FUNCTION_BLOCK Test_WhenBusy_Abort_SelectsAborting EXTENDS TUnitTestbase
VAR
END_VAR

METHOD  Execute
VAR
    Execution : TExecution;
END_VAR
Test_Started();

Execution.Start();
Execution.SetBusy();
Execution.Abort();

Assertion.AssertEquals_BOOL(
    Expected := TRUE,
    Actual   := Execution.Aborting,
    ObjectName := _TestName,
    VariableName  := 'Execution.Aborting');

Test_Finished();
END_METHOD

END_FUNCTION_BLOCK

(* stored: Version 1.1.0.1, ProductVersion 3.1.4024.3
   POU Test_WhenBusy_Abort_SelectsAborting: Id {8318710c-f8d2-4ba9-8dcc-07a00e8e1868}, SpecialFunc None
   Method Execute: Id {1d623fb4-6290-4231-8fce-d12b4af92c05} *)
